# EPICS autosave request: iocs/pilatusIOC/iocBoot/iocPilatus/auto_settings.req
file "pilatus_settings.req",      P=$(P),  R=cam1:
file "NDStdArrays_settings.req",  P=$(P),  R=image1:
file "commonPlugin_settings.req", P=$(P)
